// SIMATIC S7-200 project (STEP 7-Micro/WIN), CPU 222 CN REL 02.01

ORGANIZATION_BLOCK 主程序:OB1
TITLE=程序控制松达机械厂的裁断机，进行材料切割。
// 物理设备包括工作台、刀具、电机、安全门、启动按钮、停止按钮、紧急停止按钮和传感器。
// 操作员将材料放置在工作台上，通过按下启动按钮 启动设备。
// 主电机输出仅在启动按钮 为ON或主电机输出已为ON，且安全门传感器为ON、停止按钮为OFF时才会启动，确保设备只有在安全门关闭且未被停止时才能运行。此外，运行时安全门必须关闭，即主电机输出为ON时安全门传感器必须为ON，以保障操作员安全。
// 程序启动时，若系统初次上电且初始化完成标志为OFF，则调用子程序 HSC_INIT 初始化高速计数器。
// 为防止刀具移动超出安全范围，刀具移动下限必须保持在-10到+3之间，超出时程序会自动修正，确保刀具运行在可控范围内。若故障传感器1 或故障传感器2 触发，设备将立即停机，以防止进一步损害或安全事故。
BEGIN
Network 1 // 网络标题
// 网络注释
LD     SM0.1
AN     M0.6
CALL   HSC_INIT:SBR1
?000
Network 2
LD     SM0.0
MOVD   HC0, VD100
Network 3
LD     M0.6
MOVD   +0, SMD38
MOVB   16#C0, SMB37
HSC    0
Network 4
LD     V225.2
O      M0.6
AN     V225.3
A      Q0.0
=      M0.6
Network 5
LD     M0.6
MOVD   VD4, VD100
Network 6
LD     Q0.0
AN     Q0.2
AN     Q0.3
AN     I0.6
A      M0.1
LD     M0.0
AN     T33
AD>=   VD100, +40
OLD
=      Q0.1
Network 7
LDN    V225.3
AD=    VD4, VD100
=      M0.1
Network 8
LDD=   VD100, +0
=      M4.1
Network 9
LD     M4.1
TOF    T33, +10
Network 10
LDN    Q0.3
O      I0.7
O      M0.4
AN     I0.5
AN     M0.2
AN     Q0.1
=      Q0.2
Network 11
LDD>=  VD100, VD12
=      M0.2
Network 12
LD     I0.4
O      M0.4
AN     M0.2
AN     I0.5
=      M0.4
Network 13
LDD<=  VD100, VD8
=      M0.3
Network 14
LDD>=  VD8, +3
MOVD   +3, VD8
Network 15
LDD<=  VD8, -10
MOVD   -10, VD8
Network 16
LD     M0.0
AN     M0.4
A      Q0.0
AN     Q0.2
AN     I0.6
AN     I0.7
=      Q0.3
Network 17
LD     I0.3
O      M0.0
AN     I0.7
AN     I0.4
A      I0.2
AN     M0.3
A      Q0.0
=      M0.0
Network 18
LD     V225.0
O      Q0.0
A      I0.2
AN     V225.1
=      Q0.0
END_ORGANIZATION_BLOCK

SUBROUTINE_BLOCK HSC_INIT:SBR1
TITLE=
BEGIN
Network 1
LD     SM0.0
MOVB   16#FC, SMB37
MOVD   +0, SMD38
MOVD   +0, SMD42
HDEF   0, 9
ENI
HSC    0
END_SUBROUTINE_BLOCK

// SBR2: protected block, not included

// SBR3: protected block, not included

// SBR4: protected block, not included

// SBR5: protected block, not included

// (further data pages could not be read)
